{attribute 'qualified_only'}
{attribute 'strict'}
TYPE E_PIDOptimizationType :
(
	NoOvershoot,
	SomeOvershoot,
	PessenIntegralRule
);
END_TYPE

(* stored: Version 1.1.0.1, ProductVersion 3.1.4022.16
   DUT E_PIDOptimizationType: Id {24fbb2db-7f99-4a85-920b-5fba7f29c462} *)
